FUNCTION_BLOCK RxDoneSelector (* Basic Function Block Type *)
  (* Standard: 61499-2 *)
  (* Version 0.0, 7/16/2026, Schneider Electric, Template *)
  PACKAGE SE.Nereda;
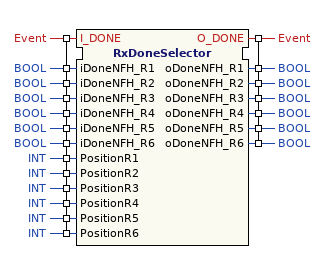
  EVENT_INPUT
    I_DONE WITH iDoneNFH_R1, iDoneNFH_R2, iDoneNFH_R3, iDoneNFH_R4, iDoneNFH_R5, iDoneNFH_R6, PositionR1, PositionR2, PositionR3, PositionR4, PositionR5, PositionR6;
  END_EVENT
  EVENT_OUTPUT
    O_DONE WITH oDoneNFH_R1, oDoneNFH_R2, oDoneNFH_R3, oDoneNFH_R4, oDoneNFH_R5, oDoneNFH_R6;
  END_EVENT
  VAR_INPUT
    iDoneNFH_R1 : BOOL;
    iDoneNFH_R2 : BOOL;
    iDoneNFH_R3 : BOOL;
    iDoneNFH_R4 : BOOL;
    iDoneNFH_R5 : BOOL;
    iDoneNFH_R6 : BOOL;
    PositionR1 : INT;
    PositionR2 : INT;
    PositionR3 : INT;
    PositionR4 : INT;
    PositionR5 : INT;
    PositionR6 : INT;
  END_VAR
  VAR_OUTPUT
    oDoneNFH_R1 : BOOL;
    oDoneNFH_R2 : BOOL;
    oDoneNFH_R3 : BOOL;
    oDoneNFH_R4 : BOOL;
    oDoneNFH_R5 : BOOL;
    oDoneNFH_R6 : BOOL;
  END_VAR
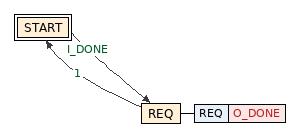
  EC_STATES
    START; (* Initial State *)
    REQ : REQ -> O_DONE; (* Normal execution *)
  END_STATES
  EC_TRANSITIONS
    START TO REQ := I_DONE;
    REQ TO START := 1;
  END_TRANSITIONS
  ALGORITHM REQ IN ST: (* Normally executed algorithm *)
;
oDoneNFH_R1 := 	(iDoneNFH_R1 AND (PositionR1 = 1)) OR
				(iDoneNFH_R2 AND (PositionR2 = 1)) OR
				(iDoneNFH_R3 AND (PositionR3 = 1)) OR
				(iDoneNFH_R4 AND (PositionR4 = 1)) OR
				(iDoneNFH_R5 AND (PositionR5 = 1)) OR
				(iDoneNFH_R6 AND (PositionR6 = 1));

oDoneNFH_R2 := 	(iDoneNFH_R1 AND (PositionR1 = 2)) OR
				(iDoneNFH_R2 AND (PositionR2 = 2)) OR
				(iDoneNFH_R3 AND (PositionR3 = 2)) OR
				(iDoneNFH_R4 AND (PositionR4 = 2)) OR
				(iDoneNFH_R5 AND (PositionR5 = 2)) OR
				(iDoneNFH_R6 AND (PositionR6 = 2));

oDoneNFH_R3 := 	(iDoneNFH_R1 AND (PositionR1 = 3)) OR
				(iDoneNFH_R2 AND (PositionR2 = 3)) OR
				(iDoneNFH_R3 AND (PositionR3 = 3)) OR
				(iDoneNFH_R4 AND (PositionR4 = 3)) OR
				(iDoneNFH_R5 AND (PositionR5 = 3)) OR
				(iDoneNFH_R6 AND (PositionR6 = 3));

oDoneNFH_R4 := 	(iDoneNFH_R1 AND (PositionR1 = 4)) OR
				(iDoneNFH_R2 AND (PositionR2 = 4)) OR
				(iDoneNFH_R3 AND (PositionR3 = 4)) OR
				(iDoneNFH_R4 AND (PositionR4 = 4)) OR
				(iDoneNFH_R5 AND (PositionR5 = 4)) OR
				(iDoneNFH_R6 AND (PositionR6 = 4));

oDoneNFH_R5 := 	(iDoneNFH_R1 AND (PositionR1 = 5)) OR
				(iDoneNFH_R2 AND (PositionR2 = 5)) OR
				(iDoneNFH_R3 AND (PositionR3 = 5)) OR
				(iDoneNFH_R4 AND (PositionR4 = 5)) OR
				(iDoneNFH_R5 AND (PositionR5 = 5)) OR
				(iDoneNFH_R6 AND (PositionR6 = 5));

oDoneNFH_R6 := 	(iDoneNFH_R1 AND (PositionR1 = 6)) OR
				(iDoneNFH_R2 AND (PositionR2 = 6)) OR
				(iDoneNFH_R3 AND (PositionR3 = 6)) OR
				(iDoneNFH_R4 AND (PositionR4 = 6)) OR
				(iDoneNFH_R5 AND (PositionR5 = 6)) OR
				(iDoneNFH_R6 AND (PositionR6 = 6));
  END_ALGORITHM
END_FUNCTION_BLOCK
